(* CODESYS project SingleElevator.project

Project tree, tasks and I/O mapping:
  Device : CODESYS Control Win V3, 3S - Smart Software Solutions GmbH, version 3.5.12.20
    application Application
      libraries: Standard, * (System)
      task MainTask (cyclic, interval 30 ms, priority 1) calls Simulation, POU, GA_Collector
      task VISU_TASK (cyclic, interval 200 ms, priority 31) calls VisuElems.Visu_Prg
      program GA_Collector [FBD]
      global variables GVL
      program POU [SFC]: Doors_Closing_Homing_exit, Doors_Opening_Homing_exit, Homing_Motor_exit, Motor_Usage_active, Doors_Closing_active, Motor_Usage_exit, Doors_Opening_exit, Internal_Panel_exit, Internal_Panel_active, Doors_Closing_exit, Doors_Opening_active, Homing_Motor_active, Doors_Opening_Homing_active, Doors_Closing_Homing_active
      GAs/
        function block Doors_GA [SFC]: Ready_active, Busy_active
        function block Call_Management_GA [SFC]: Turn_Off_5_active, Refresh_dim_log_exit, P5_exit, Turn_Off_1_active, P2_active, P7_exit, Destination_Update_exit, Turn_Off_6_active, P3_exit, Destination_OUT_active, Wait_TIME_active, Ready_active, Ready_exit, P7_active, Turn_Off_G_active, WAIT_active, PG_active, Can_Go_active, P5_active, Sorting_Int_entry, Turn_Off_7_active, P6_exit, P6_active, Turn_Off_2_active, P2_exit, Turn_Off_4_active, Wait_Start_active, Waiting_Int_active, P1_exit, Wait_TIME_entry, P3_active, Destination_Update_active, P1_active, P4_active, Turn_Off_3_active, P4_exit, Refresh_dim_log_active, Turn_Off_Leds_active, Turn_Off_Leds_exit, Sorting_Int_active, Sorting_Int_exit, Waiting_Ext_active, Waiting_Int_entry, WAIT_entry, Turn_Off_3_exit, Sorting_Ext_entry, Sorting_Ext_active, Can_Go_exit, Turn_Off_Leds_entry, Control_Int_active, Wait_Passengers_exit
        function block Motor_GA [SFC]: Motor_Activation_DOWN_active, Ready_active, Wait_Arrive_Up_entry, Go_G_Deck_active, Deck_Passed_entry, Step1_active, Busy_active, Motor_Activation_Homing_active, Go_G_Deck_exit, Arrived_UP_exit, Arrived_Down_exit, Wait_Arrive_Up_exit, Motor_Activation_UP_active, Motor_Activation_Homing_exit, Wait_Arrive_Down_exit, Motor_Activation_Homing_entry, Wait_Arrive_Down_entry
      visualisation Visualization
      program Simulation [ST]
  text list GlobalTextList
*)

// Device/Application/GVL
VAR_GLOBAL
(* Elevator managing variables*)
	Open: BOOL;				(* Sensor: the door is fully open*)
	Closed: BOOL;			(* Sensor: the door is fully closed*)
	LimitDown: BOOL;		(* Sensor: lower limit sensor, if TRUE the lift has reached the lower limit*)
	LimitUp: BOOL;			(* Sensor: upper limit sensor, if TRUE the lift has reached the upper limit*)
	DeckSensor: BOOL;		(* Sensor: if TRUE the cab is in proximity of a deck*)
	RampSensor: BOOL;		(* Sensor: if TRUE the cab is in proximity of a ramp*)
	Presence :BOOL; 		(* Sensor: if TRUE something blocks the door photocell*)
	Emergency: BOOL;		(* Input: if TRUE the emergency button has been pressed*)

	Closing: BOOL;			(* Actuator: if TRUE the door starts closing*)
	Opening: BOOL;			(* Actuator: the door starts opening*)
	Motor_on: BOOL;			(* Actuator: if TRUE the lift pulley motor start moving*)
	Up: BOOL;				(* Actuator parameter: if TRUE the lift moves upward, downward otherwise*)
	Vel: BOOL;				(* Actuator parameter: motor speed, if TRUE high speed, low speed otherwise*)


	Current: INT;  			(* Visualization: variable used to storage the current deck*)
    Destination: INT;		(* Visualization: variable used to storage the the destination deck*)
	EmergencyVis: BOOL; 	(* Visualization: if TRUE the emergency light is turned on*)

	InitialDeck: INT := 1;	(* Only for simulation: variable used to define the initial deck*)
	InitCycle: BOOL := FALSE;(* Only for simulation: used to execute the instruction at the first cycle*)
	Height: INT;			(* Only for simulation: elevator height*)
	DeckRest: INT;        	(* Only for simulation: division rest for generating deck sensor*)
	Memory: INT;
	RampRest: INT;			(* Only for simulation: division rest for generating the ramp position*)
	MemoryR: INT;
	Door: INT;				(* Only for simulation: to visualize the closing of the door*)
	Displacement: INT;		(* Only for simulation: lift displacement, dependent on the motor speed*)

 (*Inputs: internal panel variables*)
	PG: BOOL;
	P1: BOOL;
	P2: BOOL;
	P3: BOOL;
	P4: BOOL;
	P5: BOOL;
	P6: BOOL;
	P7: BOOL;

(*Visualization: internal panel variables used to turn on the LED*)
	PGVis: BOOL;
	P1Vis: BOOL;
	P2Vis: BOOL;
	P3Vis: BOOL;
	P4Vis: BOOL;
	P5Vis: BOOL;
	P6Vis: BOOL;
	P7Vis: BOOL;

(*Inputs: external panel variables*)
	UpDeckG: BOOL;
	UpDeck1: BOOL;
	UpDeck2: BOOL;
	UpDeck3: BOOL;
	UpDeck4: BOOL;
	UpDeck5: BOOL;
	UpDeck6: BOOL;
	DownDeck7: BOOL;
	DownDeck6: BOOL;
	DownDeck5: BOOL;
	DownDeck4: BOOL;
	DownDeck3: BOOL;
	DownDeck2: BOOL;
	DownDeck1: BOOL;

(*Visualization: external panel variables used to turn on the LED*)
	UpDeckGVis: BOOL;
	UpDeck1Vis: BOOL;
	UpDeck2Vis: BOOL;
	UpDeck3Vis: BOOL;
	UpDeck4Vis: BOOL;
	UpDeck5Vis: BOOL;
	UpDeck6Vis: BOOL;
	DownDeck7Vis: BOOL;
	DownDeck6Vis: BOOL;
	DownDeck5Vis: BOOL;
	DownDeck4Vis: BOOL;
	DownDeck3Vis: BOOL;
	DownDeck2Vis: BOOL;
	DownDeck1Vis: BOOL;

(*Only for simulation: variables used to simulate the fault on deck sensor*)
	SensorG: BOOL;				(* if TRUE the magnetic information for deck G is lost and the deck sensor cannot become TRUE*)
	Sensor1: BOOL;				(* if TRUE the magnetic information for deck 1 is lost and the deck sensor cannot become TRUE*)
	Sensor2: BOOL;
	Sensor3: BOOL;
	Sensor4: BOOL;
	Sensor5: BOOL;
	Sensor6: BOOL;
	Sensor7: BOOL;
	FaultSensorAlarm: BOOL; 	(* Visulaization: if TRUE alerts the user of a deck sensor fault*)

(*Only for simulation: variables used to simulate the fault on ramp sensor*)
	RampGUp: BOOL;
	Ramp1Down: BOOL;
	Ramp1Up:BOOL;
	Ramp2Down: BOOL;
	Ramp2Up:BOOL;
	Ramp3Down: BOOL;
	Ramp3Up:BOOL;
	Ramp4Down: BOOL;
	Ramp4Up:BOOL;
	Ramp5Down: BOOL;
	Ramp5Up:BOOL;
	Ramp6Down: BOOL;
	Ramp6Up:BOOL;
	Ramp7Down: BOOL;
	FaultRampAlarm: BOOL; 		(* Visulaization: if TRUE alerts the user of a ramp sensor fault*)
	SensorGOK: BOOL;
	Sensor1OK: BOOL;
	Sensor2OK: BOOL;
	Sensor6OK: BOOL;
	Sensor3OK: BOOL;
	Sensor4OK: BOOL;
	Sensor5OK: BOOL;
	Sensor7OK: BOOL;
	RampGUpOK: BOOL;
	Ramp1DownOK: BOOL;
	Ramp1UpOK: BOOL;
	Ramp2DownOK: BOOL;
	Ramp2UpOK: BOOL;
	Ramp3DownOK: BOOL;
	Ramp3UpOK: BOOL;
	Ramp4DownOK: BOOL;
	Ramp4UpOK: BOOL;
	Ramp5DownOK: BOOL;
	Ramp5UpOK: BOOL;
	Ramp6DownOK: BOOL;
	Ramp6UpOK: BOOL;
	Ramp7DownOK: BOOL;
	Ramp7UpOK: BOOL;
	Doors: Doors_GA;
	Motor: Motor_GA;
	Call_Management: Call_Management_GA;
END_VAR

// Device/Application/Simulation
PROGRAM Simulation
VAR
END_VAR

(* Initial position of the cab inside the hoistway. It is executed only at the first cycle.  *)
IF NOT GVL.InitCycle THEN
			GVL.InitCycle := TRUE ;
			GVL.Height := 20 * GVL.InitialDeck;
		    GVL.Door := 0;
			GVL.Current := GVL.Height / 20;
END_IF;

(* Elevator management, these instructions are executed each cycle time*)

(* Elevator door control. *)
IF GVL.Closing THEN
	GVL.Door := GVL.Door + 1;		(*Closing door management*)
	GVL.Open := FALSE;
END_IF

IF GVL.Door >= 60 THEN						(* Closed door limit*)
	GVL.Closed := TRUE;
END_IF

IF GVL.Opening THEN
	GVL.Door := GVL.Door - 1; 	(* Opening door management*)
	GVL.Closed := FALSE;
END_IF

IF GVL.Door <= 0 THEN							(* Open door limit*)
	GVL.Open := TRUE;
END_IF


(* Maximum and minimum management in the door simulation*)
IF GVL.Door < 0 THEN
	 GVL.Door := 0;
END_IF

IF GVL.Door > 60 THEN
	GVL.Door := 60;
END_IF


(* Control of the cab position inside the hostway. *)
(* Displacement definition for graphic visualization*)
IF GVL.Vel THEN 
	GVL.Displacement := 2;
ELSE 
	GVL.Displacement := 1;
END_IF


(* Height modification relying on direction and speed*)
IF GVL.Motor_on AND GVL.Up THEN
	GVL.Height := GVL.Height + GVL.Displacement;
	GVL.LimitDown := FALSE;
END_IF

IF GVL.Motor_on AND NOT GVL.Up THEN
	GVL.Height := GVL.Height - GVL.Displacement;
	GVL.LimitUp := FALSE;
END_IF


(* Limits for visualization*)
IF GVL.Height < -20 THEN
	GVL.Height := -20;
END_IF

IF GVL.Height > 160 THEN
	GVL.Height := 160;
END_IF

(* Limit sensors management*)
IF GVL.Height <= -10 THEN
	GVL.LimitDown := TRUE;
END_IF

IF GVL.Height >= 150 THEN
	 GVL.LimitUp := TRUE;
END_IF


(*-------------------------------------------------------------------*)
(*  Fault Management (Deck and Ramp Sensors)   *)
(*-------------------------------------------------------------------*)
(* Deck Sensor*)
(* Range of value where the deck sensor is active*)
IF ((GVL.Height >= -1) AND (GVL.Height <= 1)) THEN
	GVL.SensorGOK := TRUE;
ELSE  
	GVL.SensorGOK := FALSE;
END_IF

IF ((GVL.Height >= 20-1) AND (GVL.Height <= 20+1)) THEN
	GVL.Sensor1OK := TRUE;
ELSE  
	GVL.Sensor1OK := FALSE;
END_IF

IF ((GVL.Height >= 40-1) AND (GVL.Height <= 40+1)) THEN
	GVL.Sensor2OK := TRUE;
ELSE  
	GVL.Sensor2OK := FALSE;
END_IF

IF ((GVL.Height >= 60-1) AND (GVL.Height <= 60+1)) THEN
	GVL.Sensor3OK := TRUE;
ELSE  
	GVL.Sensor3OK := FALSE;
END_IF

IF ((GVL.Height >= 80-1) AND (GVL.Height <= 80+1)) THEN
	GVL.Sensor4OK := TRUE;
ELSE  
	GVL.Sensor4OK := FALSE;
END_IF

IF ((GVL.Height >= 100-1) AND (GVL.Height <= 100+1)) THEN
	GVL.Sensor5OK := TRUE;
ELSE   
	GVL.Sensor5OK := FALSE;
END_IF

IF ((GVL.Height >= 120-1) AND (GVL.Height <= 120+1)) THEN
	GVL.Sensor6OK := TRUE;
ELSE  
	GVL.Sensor6OK := FALSE;
END_IF

IF ((GVL.Height >= 140-1) AND (GVL.Height <= 140+1)) THEN
	GVL.Sensor7OK := TRUE;
ELSE  
	GVL.Sensor7OK := FALSE;
END_IF

GVL.DeckSensor := (GVL.SensorGOK AND NOT GVL.SensorG) OR
				    (GVL.Sensor1OK AND NOT GVL.Sensor1) OR
				    (GVL.Sensor2OK AND NOT GVL.Sensor2) OR
				    (GVL.Sensor3OK AND NOT GVL.Sensor3) OR
				    (GVL.Sensor4OK AND NOT GVL.Sensor4) OR
				    (GVL.Sensor5OK AND NOT GVL.Sensor5) OR
				    (GVL.Sensor6OK AND NOT GVL.Sensor6) OR
				    (GVL.Sensor7OK AND NOT GVL.Sensor7);

(* Ramp Sensor*)
(* Range of value where the ramp sensor is active*)
IF ((GVL.Height >= 5-1) AND (GVL.Height <= 5+1)) THEN
	GVL.RampGUpOK := TRUE;
ELSE 
	GVL.RampGUpOK := FALSE;
END_IF

(* Ramp close to deck 1*)
IF ((GVL.Height >= 15-1) AND (GVL.Height <= 15+1)) THEN
	GVL.Ramp1DownOK := TRUE;
ELSE 
	GVL.Ramp1DownOK := FALSE;
END_IF

IF ((GVL.Height >= 25-1) AND (GVL.Height <= 25+1)) THEN
	GVL.Ramp1UpOK := TRUE;
ELSE 
	GVL.Ramp1UpOK := FALSE;
END_IF

(* Ramp close to deck 2*)
IF ((GVL.Height >= 35-1) AND (GVL.Height <= 35+1)) THEN
	GVL.Ramp2DownOK := TRUE;
ELSE 
	GVL.Ramp2DownOK := FALSE;
END_IF

IF ((GVL.Height >= 45-1) AND (GVL.Height <= 45+1)) THEN
	GVL.Ramp2UpOK := TRUE;
ELSE 
	GVL.Ramp2UpOK := FALSE;
END_IF

(*Ramp close to deck  3*)
IF ((GVL.Height >= 55-1) AND (GVL.Height <= 55+1)) THEN
	GVL.Ramp3DownOK := TRUE;
ELSE 
	GVL.Ramp3DownOK := FALSE;
END_IF

IF ((GVL.Height >= 65-1) AND (GVL.Height <= 65+1)) THEN
	GVL.Ramp3UpOK := TRUE;
ELSE 
	GVL.Ramp3UpOK := FALSE;
END_IF

(* Ramp close to deck  4*)
IF ((GVL.Height >= 75-1) AND (GVL.Height <= 75+1)) THEN
	GVL.Ramp4DownOK := TRUE;
ELSE 
	GVL.Ramp4DownOK := FALSE;
END_IF

IF ((GVL.Height >= 85-1) AND (GVL.Height <= 85+1)) THEN
	GVL.Ramp4UpOK := TRUE;
ELSE 
	GVL.Ramp4UpOK:=FALSE;
END_IF

(* Ramp close to deck  5*)
IF ((GVL.Height >= 95-1) AND (GVL.Height <= 95+1)) THEN
	GVL.Ramp5DownOK := TRUE;
ELSE 
	GVL.Ramp5DownOK := FALSE;
END_IF

IF ((GVL.Height >= 105-1) AND (GVL.Height <= 105+1)) THEN
	GVL.Ramp5UpOK := TRUE;
ELSE
	GVL.Ramp5UpOK := FALSE;
END_IF

(* Ramp close to deck  6*)
IF ((GVL.Height >= 115-1) AND (GVL.Height <= 115+1)) THEN
	GVL.Ramp6DownOK := TRUE;
ELSE 
	GVL.Ramp6DownOK := FALSE;
END_IF

IF ((GVL.Height >= 125-1) AND (GVL.Height <= 125+1)) THEN
	GVL.Ramp6UpOK := TRUE;
ELSE 
	GVL.Ramp6UpOK := FALSE;
END_IF

(* Ramp close to deck  7*)
IF ((GVL.Height >= 135-1) AND (GVL.Height <= 135+1)) THEN
	GVL.Ramp7DownOK := TRUE;
ELSE 
	GVL.Ramp7DownOK := FALSE;
END_IF

GVL.RampSensor:=(GVL.RampGUpOK AND NOT GVL.RampGUp) OR 
								(GVL.Ramp1DownOK AND NOT GVL.Ramp1Down ) OR 
								(GVL.Ramp1UpOK AND NOT GVL.Ramp1Up ) OR
								(GVL.Ramp2DownOK AND NOT GVL.Ramp2Down ) OR 
								(GVL.Ramp2UpOK AND NOT GVL.Ramp2Up ) OR
								(GVL.Ramp3DownOK AND NOT GVL.Ramp3Down ) OR
 								(GVL.Ramp3UpOK AND NOT GVL.Ramp3Up ) OR
								(GVL.Ramp4DownOK AND NOT GVL.Ramp4Down ) OR
 								(GVL.Ramp4UpOK AND NOT GVL.Ramp4Up ) OR
								(GVL.Ramp5DownOK AND NOT GVL.Ramp5Down ) OR
 								(GVL.Ramp5UpOK AND NOT GVL.Ramp5Up ) OR
								(GVL.Ramp6DownOK AND NOT GVL.Ramp6Down ) OR
								(GVL.Ramp6UpOK AND NOT GVL.Ramp6Up ) OR
								(GVL.Ramp7DownOK AND NOT GVL.Ramp7Down );

END_PROGRAM

// Device/Application/POU
PROGRAM POU
VAR
	Operation_OK: BOOL;
	Synchronization : BOOL;
END_VAR

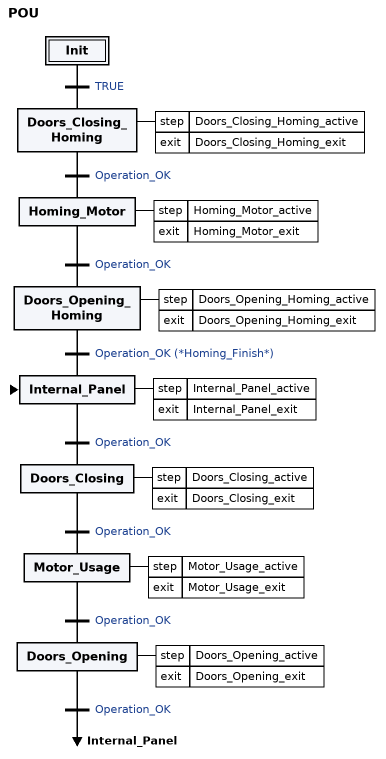
INITIAL_STEP Init:
END_STEP
TRANSITION FROM Init TO Doors_Closing_Homing
    := TRUE;
END_TRANSITION
STEP Doors_Closing_Homing:
    Doors_Closing_Homing_active(N);  // step action
    Doors_Closing_Homing_exit(P0);  // exit action
END_STEP
TRANSITION FROM Doors_Closing_Homing TO Homing_Motor
    := Operation_OK;
END_TRANSITION
STEP Homing_Motor:
    Homing_Motor_active(N);  // step action
    Homing_Motor_exit(P0);  // exit action
END_STEP
TRANSITION FROM Homing_Motor TO Doors_Opening_Homing
    := Operation_OK;
END_TRANSITION
STEP Doors_Opening_Homing:
    Doors_Opening_Homing_active(N);  // step action
    Doors_Opening_Homing_exit(P0);  // exit action
END_STEP
TRANSITION FROM Doors_Opening_Homing TO Internal_Panel
    := Operation_OK (*Homing_Finish*);
END_TRANSITION
STEP Internal_Panel:
    Internal_Panel_active(N);  // step action
    Internal_Panel_exit(P0);  // exit action
END_STEP
TRANSITION FROM Internal_Panel TO Doors_Closing
    := Operation_OK;
END_TRANSITION
STEP Doors_Closing:
    Doors_Closing_active(N);  // step action
    Doors_Closing_exit(P0);  // exit action
END_STEP
TRANSITION FROM Doors_Closing TO Motor_Usage
    := Operation_OK;
END_TRANSITION
STEP Motor_Usage:
    Motor_Usage_active(N);  // step action
    Motor_Usage_exit(P0);  // exit action
END_STEP
TRANSITION FROM Motor_Usage TO Doors_Opening
    := Operation_OK;
END_TRANSITION
STEP Doors_Opening:
    Doors_Opening_active(N);  // step action
    Doors_Opening_exit(P0);  // exit action
END_STEP
TRANSITION FROM Doors_Opening TO Internal_Panel
    := Operation_OK;
END_TRANSITION

ACTION Doors_Closing_Homing_exit:
Operation_OK:=FALSE;
Synchronization:=FALSE;
END_ACTION

ACTION Doors_Opening_Homing_exit:
Operation_OK:=FALSE;
Synchronization:=FALSE;
END_ACTION

ACTION Homing_Motor_exit:
Operation_OK:=FALSE;
Synchronization:=FALSE;
END_ACTION

ACTION Motor_Usage_active:
IF Motor.State = 'Ready' THEN
	Motor.Do_:= TRUE;
	Motor.STOP := FALSE;
	IF ( Call_Management.Destination_Deck[0] > Current AND Call_Management.Destination_Deck[0] <> 8 ) THEN
		Motor.Do_What := 'Go_Up';
	END_IF
	IF ( Call_Management.Destination_Deck[0] < Current AND Call_Management.Destination_Deck[0] <> 8 ) THEN
		Motor.Do_What := 'Go_Down';
	END_IF
END_IF

IF (Motor.State = 'Busy' AND Current = Call_Management.Destination_Deck [0] - 1 AND Motor.Do_What = 'Go_Up' OR Call_Management.Destination_Deck [0] = 8 ) THEN;
	Motor.STOP := TRUE;	
END_IF

IF (Motor.State = 'Busy' AND Current = Call_Management.Destination_Deck [0] + 1 AND Motor.Do_What = 'Go_Down' OR Call_Management.Destination_Deck [0] = 8 ) THEN;
	Motor.STOP := TRUE;	
END_IF

IF Motor.State = 'Busy' AND Motor.Done = TRUE THEN
	Motor.Do_ := FALSE;
	Motor.STOP := FALSE;
	Synchronization := TRUE;
END_IF

Operation_OK := Synchronization AND NOT Motor.Done;
END_ACTION

ACTION Doors_Closing_active:
IF Doors.State = 'Ready' THEN
	Doors.Do_:= TRUE;
	Doors.Do_what := 'Close';
END_IF

IF Doors.State = 'Busy' AND Doors.Done = TRUE THEN
	Doors.Do_ := FALSE;
	Synchronization := TRUE;
END_IF

Operation_OK := Synchronization AND NOT Doors.Done;
END_ACTION

ACTION Motor_Usage_exit:
Operation_OK:=FALSE;
Synchronization:=FALSE;
END_ACTION

ACTION Doors_Opening_exit:
Operation_OK:=FALSE;
Synchronization:=FALSE;
END_ACTION

ACTION Internal_Panel_exit:
Operation_OK:=FALSE;
Synchronization:=FALSE;
END_ACTION

ACTION Internal_Panel_active:
IF Call_Management.State = 'Ready' THEN
	Call_Management.Start:= TRUE;
	Call_Management.Stop:= FALSE;
END_IF

IF Call_Management.State = 'Can_Go' THEN
	Synchronization := TRUE;
END_IF

Operation_OK := Synchronization;
END_ACTION

ACTION Doors_Closing_exit:
Operation_OK:=FALSE;
Synchronization:=FALSE;
END_ACTION

ACTION Doors_Opening_active:
IF Doors.State = 'Ready' THEN
	Doors.Do_:= TRUE;
	Doors.Do_what := 'Open';
END_IF

IF Doors.State = 'Busy' AND Doors.Done = TRUE AND Call_Management.Destination_Deck[0] <> 8 THEN
	Doors.Do_ := FALSE;
	Synchronization := TRUE;
END_IF

Operation_OK := Synchronization AND NOT Doors.Done;
END_ACTION

ACTION Homing_Motor_active:
IF Motor.State = 'Ready' THEN
	Motor.Do_:= TRUE;
	Motor.Do_What := 'Homing';
END_IF

IF Motor.State = 'Busy' AND Motor.Done = TRUE THEN
	Motor.Do_ := FALSE;
	Synchronization := TRUE;
END_IF

Operation_OK := Synchronization AND NOT Motor.Done;
END_ACTION

ACTION Doors_Opening_Homing_active:
IF Doors.State = 'Ready' THEN
	Doors.Do_:= TRUE;
	Doors.Do_what := 'Open';
END_IF

IF Doors.State = 'Busy' AND Doors.Done = TRUE THEN
	Doors.Do_ := FALSE;
	Synchronization := TRUE;
END_IF

Operation_OK := Synchronization AND NOT Doors.Done;
END_ACTION

ACTION Doors_Closing_Homing_active:
IF Doors.State = 'Ready' THEN
	Doors.Do_:= TRUE;
	Doors.Do_what := 'Close';
END_IF

IF Doors.State = 'Busy' AND Doors.Done = TRUE THEN
	Doors.Do_ := FALSE;
	Synchronization := TRUE;
END_IF

Operation_OK := Synchronization AND NOT Doors.Done;
END_ACTION

END_PROGRAM

// Device/Application/GA_Collector
PROGRAM GA_Collector
VAR
END_VAR

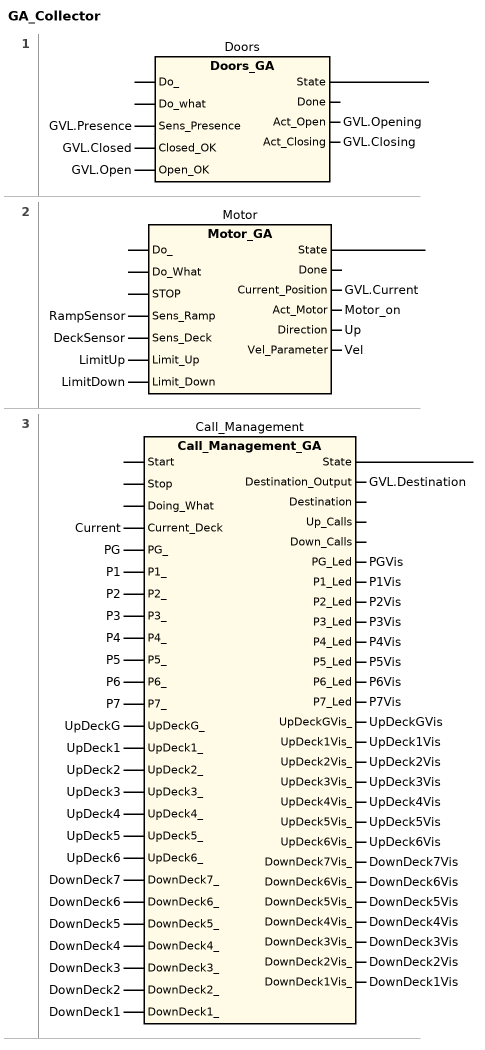
// NETWORK 1
Doors(
    Sens_Presence := GVL.Presence,
    Closed_OK := GVL.Closed,
    Open_OK := GVL.Open,
    Act_Open => GVL.Opening,
    Act_Closing => GVL.Closing); // Doors_GA

// NETWORK 2
Motor(
    Sens_Ramp := RampSensor,
    Sens_Deck := DeckSensor,
    Limit_Up := LimitUp,
    Limit_Down := LimitDown,
    Current_Position => GVL.Current,
    Act_Motor => Motor_on,
    Direction => Up,
    Vel_Parameter => Vel); // Motor_GA

// NETWORK 3
Call_Management(
    Current_Deck := Current,
    PG_ := PG,
    P1_ := P1,
    P2_ := P2,
    P3_ := P3,
    P4_ := P4,
    P5_ := P5,
    P6_ := P6,
    P7_ := P7,
    UpDeckG_ := UpDeckG,
    UpDeck1_ := UpDeck1,
    UpDeck2_ := UpDeck2,
    UpDeck3_ := UpDeck3,
    UpDeck4_ := UpDeck4,
    UpDeck5_ := UpDeck5,
    UpDeck6_ := UpDeck6,
    DownDeck7_ := DownDeck7,
    DownDeck6_ := DownDeck6,
    DownDeck5_ := DownDeck5,
    DownDeck4_ := DownDeck4,
    DownDeck3_ := DownDeck3,
    DownDeck2_ := DownDeck2,
    DownDeck1_ := DownDeck1,
    Destination_Output => GVL.Destination,
    PG_Led => PGVis,
    P1_Led => P1Vis,
    P2_Led => P2Vis,
    P3_Led => P3Vis,
    P4_Led => P4Vis,
    P5_Led => P5Vis,
    P6_Led => P6Vis,
    P7_Led => P7Vis,
    UpDeckGVis_ => UpDeckGVis,
    UpDeck1Vis_ => UpDeck1Vis,
    UpDeck2Vis_ => UpDeck2Vis,
    UpDeck3Vis_ => UpDeck3Vis,
    UpDeck4Vis_ => UpDeck4Vis,
    UpDeck5Vis_ => UpDeck5Vis,
    UpDeck6Vis_ => UpDeck6Vis,
    DownDeck7Vis_ => DownDeck7Vis,
    DownDeck6Vis_ => DownDeck6Vis,
    DownDeck5Vis_ => DownDeck5Vis,
    DownDeck4Vis_ => DownDeck4Vis,
    DownDeck3Vis_ => DownDeck3Vis,
    DownDeck2Vis_ => DownDeck2Vis,
    DownDeck1Vis_ => DownDeck1Vis); // Call_Management_GA

END_PROGRAM

// Device/Application/GAs/Doors_GA
FUNCTION_BLOCK Doors_GA
VAR_INPUT
	Do_: BOOL;
	Do_what: STRING;
	Sens_Presence: BOOL;
	Closed_OK: BOOL;
	Open_OK: BOOL;
END_VAR
VAR_OUTPUT
	State: STRING;
	Done: BOOL;
	Act_Open: BOOL;
	Act_Closing: BOOL;
END_VAR
VAR	
END_VAR

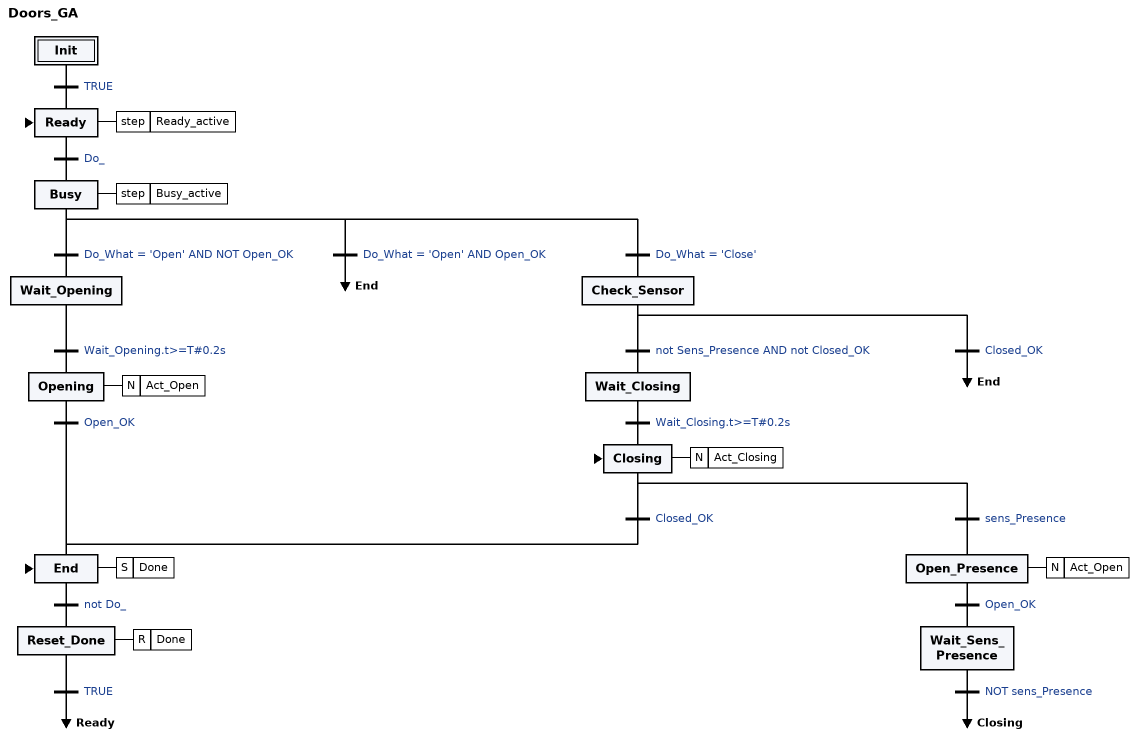
INITIAL_STEP Init:
END_STEP
TRANSITION FROM Init TO Ready
    := TRUE;
END_TRANSITION
STEP Ready:
    Ready_active(N);  // step action
END_STEP
TRANSITION FROM Ready TO Busy
    := Do_;
END_TRANSITION
STEP Busy:
    Busy_active(N);  // step action
END_STEP
TRANSITION FROM Busy TO Wait_Opening
    := Do_What = 'Open' AND NOT Open_OK;
END_TRANSITION
STEP Wait_Opening:
END_STEP
TRANSITION FROM Wait_Opening TO Opening
    := Wait_Opening.t>=T#0.2s;
END_TRANSITION
STEP Opening:
    Act_Open(N);
END_STEP
TRANSITION FROM Opening TO End
    := Open_OK;
END_TRANSITION
TRANSITION FROM Busy TO End
    := Do_What = 'Open' AND Open_OK;
END_TRANSITION
TRANSITION FROM Busy TO Check_Sensor
    := Do_What = 'Close';
END_TRANSITION
STEP Check_Sensor:
END_STEP
TRANSITION FROM Check_Sensor TO Wait_Closing
    := not Sens_Presence AND not Closed_OK;
END_TRANSITION
STEP Wait_Closing:
END_STEP
TRANSITION FROM Wait_Closing TO Closing
    := Wait_Closing.t>=T#0.2s;
END_TRANSITION
STEP Closing:
    Act_Closing(N);
END_STEP
TRANSITION FROM Closing TO End
    := Closed_OK;
END_TRANSITION
TRANSITION FROM Closing TO Open_Presence
    := sens_Presence;
END_TRANSITION
STEP Open_Presence:
    Act_Open(N);
END_STEP
TRANSITION FROM Open_Presence TO Wait_Sens_Presence
    := Open_OK;
END_TRANSITION
STEP Wait_Sens_Presence:
END_STEP
TRANSITION FROM Wait_Sens_Presence TO Closing
    := NOT sens_Presence;
END_TRANSITION
TRANSITION FROM Check_Sensor TO End
    := Closed_OK;
END_TRANSITION
STEP End:
    Done(S);
END_STEP
TRANSITION FROM End TO Reset_Done
    := not Do_;
END_TRANSITION
STEP Reset_Done:
    Done(R);
END_STEP
TRANSITION FROM Reset_Done TO Ready
    := TRUE;
END_TRANSITION

ACTION Ready_active:
State := 'Ready';
END_ACTION

ACTION Busy_active:
State := 'Busy';
END_ACTION

END_FUNCTION_BLOCK

// Device/Application/GAs/Motor_GA
FUNCTION_BLOCK Motor_GA
VAR_INPUT
	Do_ : BOOL;
	Do_What: STRING;
	STOP: BOOL;
	Sens_Ramp: BOOL;
	Sens_Deck: BOOL;
	Limit_Up: BOOL;
	Limit_Down: BOOL;
END_VAR
VAR_OUTPUT
	State : STRING;
	Done : BOOL;
	Current_Position : INT;
	Act_Motor: BOOL;
	Direction: BOOL;
	Vel_Parameter: BOOL;
END_VAR
VAR
END_VAR

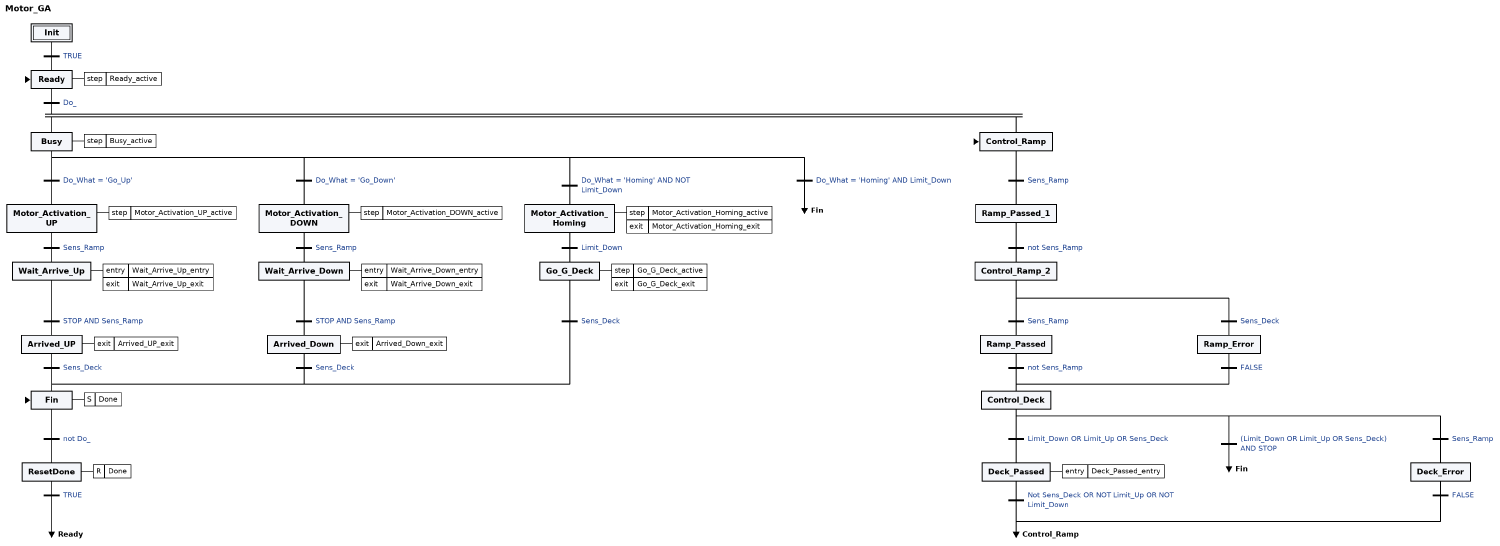
INITIAL_STEP Init:
END_STEP
TRANSITION FROM Init TO Ready
    := TRUE;
END_TRANSITION
STEP Ready:
    Ready_active(N);  // step action
END_STEP
TRANSITION FROM Ready TO (Busy, Control_Ramp)
    := Do_;
END_TRANSITION
STEP Busy:
    Busy_active(N);  // step action
END_STEP
TRANSITION FROM Busy TO Motor_Activation_UP
    := Do_What = 'Go_Up';
END_TRANSITION
STEP Motor_Activation_UP:
    Motor_Activation_UP_active(N);  // step action
END_STEP
TRANSITION FROM Motor_Activation_UP TO Wait_Arrive_Up
    := Sens_Ramp;
END_TRANSITION
STEP Wait_Arrive_Up:
    Wait_Arrive_Up_entry(P1);  // entry action
    Wait_Arrive_Up_exit(P0);  // exit action
END_STEP
TRANSITION FROM Wait_Arrive_Up TO Arrived_UP
    := STOP AND Sens_Ramp;
END_TRANSITION
STEP Arrived_UP:
    Arrived_UP_exit(P0);  // exit action
END_STEP
TRANSITION FROM Arrived_UP TO Fin
    := Sens_Deck;
END_TRANSITION
TRANSITION FROM Busy TO Motor_Activation_DOWN
    := Do_What = 'Go_Down';
END_TRANSITION
STEP Motor_Activation_DOWN:
    Motor_Activation_DOWN_active(N);  // step action
END_STEP
TRANSITION FROM Motor_Activation_DOWN TO Wait_Arrive_Down
    := Sens_Ramp;
END_TRANSITION
STEP Wait_Arrive_Down:
    Wait_Arrive_Down_entry(P1);  // entry action
    Wait_Arrive_Down_exit(P0);  // exit action
END_STEP
TRANSITION FROM Wait_Arrive_Down TO Arrived_Down
    := STOP AND Sens_Ramp;
END_TRANSITION
STEP Arrived_Down:
    Arrived_Down_exit(P0);  // exit action
END_STEP
TRANSITION FROM Arrived_Down TO Fin
    := Sens_Deck;
END_TRANSITION
TRANSITION FROM Busy TO Motor_Activation_Homing
    := Do_What = 'Homing' AND NOT Limit_Down;
END_TRANSITION
STEP Motor_Activation_Homing:
    Motor_Activation_Homing_active(N);  // step action
    Motor_Activation_Homing_exit(P0);  // exit action
END_STEP
TRANSITION FROM Busy TO Fin
    := Do_What = 'Homing' AND Limit_Down;
END_TRANSITION
TRANSITION FROM Motor_Activation_Homing TO Go_G_Deck
    := Limit_Down;
END_TRANSITION
STEP Go_G_Deck:
    Go_G_Deck_active(N);  // step action
    Go_G_Deck_exit(P0);  // exit action
END_STEP
TRANSITION FROM Go_G_Deck TO Fin
    := Sens_Deck;
END_TRANSITION
STEP Fin:
    Done(S);
END_STEP
STEP Control_Ramp:
END_STEP
TRANSITION FROM Control_Ramp TO Ramp_Passed_1
    := Sens_Ramp;
END_TRANSITION
STEP Ramp_Passed_1:
END_STEP
TRANSITION FROM Ramp_Passed_1 TO Control_Ramp_2
    := not Sens_Ramp;
END_TRANSITION
STEP Control_Ramp_2:
END_STEP
TRANSITION FROM Control_Ramp_2 TO Ramp_Passed
    := Sens_Ramp;
END_TRANSITION
STEP Ramp_Passed:
END_STEP
TRANSITION FROM Ramp_Passed TO Control_Deck
    := not Sens_Ramp;
END_TRANSITION
TRANSITION FROM Control_Ramp_2 TO Ramp_Error
    := Sens_Deck;
END_TRANSITION
STEP Ramp_Error:
END_STEP
TRANSITION FROM Ramp_Error TO Control_Deck
    := FALSE;
END_TRANSITION
STEP Control_Deck:
END_STEP
TRANSITION FROM Control_Deck TO Deck_Passed
    := Limit_Down OR Limit_Up OR Sens_Deck;
END_TRANSITION
STEP Deck_Passed:
    Deck_Passed_entry(P1);  // entry action
END_STEP
TRANSITION FROM Deck_Passed TO Control_Ramp
    := Not Sens_Deck OR NOT Limit_Up OR NOT Limit_Down;
END_TRANSITION
TRANSITION FROM Control_Deck TO Fin
    := (Limit_Down OR Limit_Up OR Sens_Deck) AND STOP;
END_TRANSITION
TRANSITION FROM Control_Deck TO Deck_Error
    := Sens_Ramp;
END_TRANSITION
STEP Deck_Error:
END_STEP
TRANSITION FROM Deck_Error TO Control_Ramp
    := FALSE;
END_TRANSITION
TRANSITION FROM Fin TO ResetDone
    := not Do_;
END_TRANSITION
STEP ResetDone:
    Done(R);
END_STEP
TRANSITION FROM ResetDone TO Ready
    := TRUE;
END_TRANSITION
// branch label Fault

ACTION Motor_Activation_DOWN_active:
Act_Motor := TRUE;
END_ACTION

ACTION Ready_active:
State := 'Ready';
END_ACTION

ACTION Wait_Arrive_Up_entry:
Vel_Parameter := TRUE;
END_ACTION

ACTION Go_G_Deck_active:
Current_Position := -1;
Direction:= TRUE;
END_ACTION

ACTION Deck_Passed_entry:
IF Do_What = 'Go_Up' AND Act_Motor THEN
	Current_Position := Current_Position +1;
END_IF

IF Do_What = 'Go_Down' AND Act_Motor THEN
	Current_Position := Current_Position -1;
END_IF
END_ACTION

ACTION Step1_active:
Current_Position := Current_Position +1;
END_ACTION

ACTION Busy_active:
State := 'Busy';
END_ACTION

ACTION Motor_Activation_Homing_active:
Act_Motor := TRUE;
(* La simulazione ha gia impostato all'interno di settare il current a -1 *)
END_ACTION

ACTION Go_G_Deck_exit:
Act_Motor := FALSE;
END_ACTION

ACTION Arrived_UP_exit:
Act_Motor := FALSE;
Direction := FALSE;
Current_Position := Current_Position +1;
END_ACTION

ACTION Arrived_Down_exit:
Act_Motor := FALSE;
Direction := FALSE;
Current_Position:= Current_Position -1;
END_ACTION

ACTION Wait_Arrive_Up_exit:
Vel_Parameter := FALSE;
END_ACTION

ACTION Motor_Activation_UP_active:
Act_Motor := TRUE;
Direction := TRUE;
END_ACTION

ACTION Motor_Activation_Homing_exit:
Current_Position := -1;
END_ACTION

ACTION Wait_Arrive_Down_exit:
Vel_Parameter := FALSE;
END_ACTION

ACTION Motor_Activation_Homing_entry:
Current_Position := 1;
END_ACTION

ACTION Wait_Arrive_Down_entry:
Vel_Parameter := TRUE;
END_ACTION

END_FUNCTION_BLOCK

// Device/Application/GAs/Call_Management_GA
FUNCTION_BLOCK Call_Management_GA
VAR_INPUT
	Start : BOOL;
	Stop: BOOL;
	Doing_What : STRING;
	Current_Deck : INT;
	PG_: BOOL; 
	P1_: BOOL;
	P2_: BOOL;
	P3_: BOOL;
	P4_: BOOL;
	P5_: BOOL;
	P6_: BOOL;
	P7_: BOOL;
	UpDeckG_: BOOL;
	UpDeck1_: BOOL;
	UpDeck2_: BOOL;
	UpDeck3_: BOOL;
	UpDeck4_: BOOL;
	UpDeck5_: BOOL;
	UpDeck6_: BOOL;
	DownDeck7_: BOOL;
	DownDeck6_: BOOL;
	DownDeck5_: BOOL;
	DownDeck4_: BOOL;
	DownDeck3_: BOOL;
	DownDeck2_: BOOL;
	DownDeck1_: BOOL;
END_VAR
VAR_OUTPUT
	State : STRING;
	Destination_Output : INT;
	Destination_Deck : ARRAY [0..7] OF INT := [8(8)];
	Up_Calls : ARRAY [0..13] OF INT := [14(8)];
	Down_Calls : ARRAY [0..13] OF INT := [14(8)];
	PG_Led: BOOL;
	P1_Led: BOOL;
	P2_Led: BOOL;
	P3_Led: BOOL;
	P4_Led: BOOL;
	P5_Led: BOOL;
	P6_Led: BOOL;
	P7_Led: BOOL;
	UpDeckGVis_: BOOL;
	UpDeck1Vis_: BOOL;
	UpDeck2Vis_: BOOL;
	UpDeck3Vis_: BOOL;
	UpDeck4Vis_: BOOL;
	UpDeck5Vis_: BOOL;
	UpDeck6Vis_: BOOL;
	DownDeck7Vis_: BOOL;
	DownDeck6Vis_: BOOL;
	DownDeck5Vis_: BOOL;
	DownDeck4Vis_: BOOL;
	DownDeck3Vis_: BOOL;
	DownDeck2Vis_: BOOL;
	DownDeck1Vis_: BOOL;
END_VAR
VAR
	{*INTERNAL PANEL SORT*}
	i : INT := 0;
	dim_cabin: INT :=0;
	j: INT;
	Sorted: BOOL;
	t: INT;
	
	{*EXTERNAL PANEL*}
	ext: INT :=0;
	z: INT;
	Position_Ext: INT :=8;
	
	k: INT :=0;
	Served: BOOL;
	
	Turned_Off: BOOL;
	Pressed_Int: BOOL;
	Pressed_Start: BOOL;
	
	g: INT;
	Finish: BOOL;
	Upgrading: BOOL;
	Upgraded: BOOL;
END_VAR

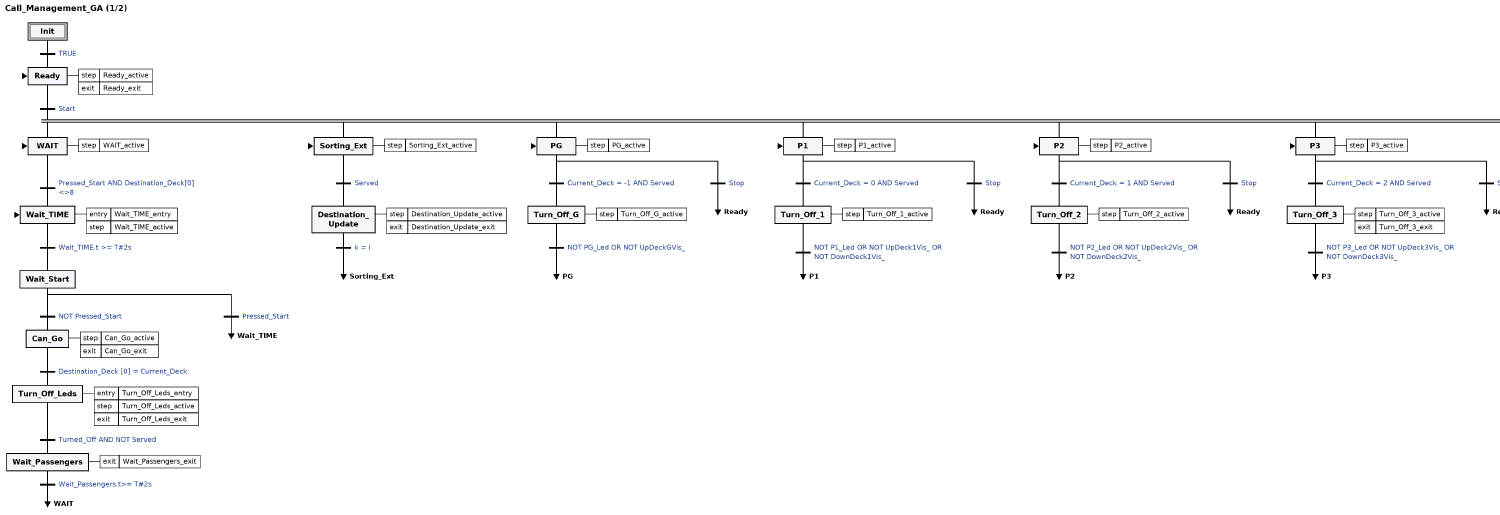
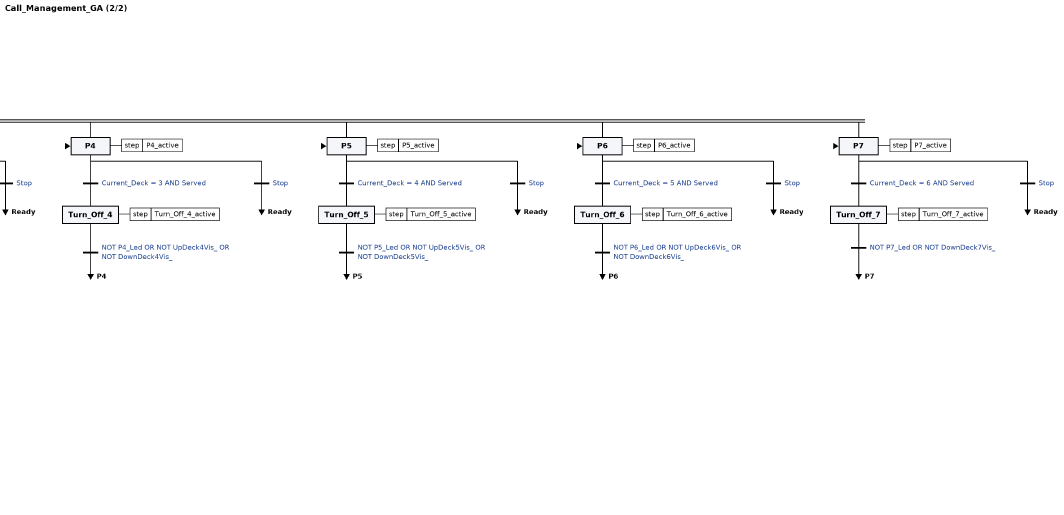
INITIAL_STEP Init:
END_STEP
TRANSITION FROM Init TO Ready
    := TRUE;
END_TRANSITION
STEP Ready:
    Ready_active(N);  // step action
    Ready_exit(P0);  // exit action
END_STEP
TRANSITION FROM Ready TO (WAIT, Sorting_Ext, PG, P1, P2, P3, P4, P5, P6, P7)
    := Start;
END_TRANSITION
STEP WAIT:
    WAIT_active(N);  // step action
END_STEP
TRANSITION FROM WAIT TO Wait_TIME
    := Pressed_Start AND Destination_Deck[0] <>8;
END_TRANSITION
STEP Wait_TIME:
    Wait_TIME_entry(P1);  // entry action
    Wait_TIME_active(N);  // step action
END_STEP
TRANSITION FROM Wait_TIME TO Wait_Start
    := Wait_TIME.t >= T#2s;
END_TRANSITION
STEP Wait_Start:
END_STEP
TRANSITION FROM Wait_Start TO Can_Go
    := NOT Pressed_Start;
END_TRANSITION
TRANSITION FROM Wait_Start TO Wait_TIME
    := Pressed_Start;
END_TRANSITION
STEP Can_Go:
    Can_Go_active(N);  // step action
    Can_Go_exit(P0);  // exit action
END_STEP
TRANSITION FROM Can_Go TO Turn_Off_Leds
    := Destination_Deck [0] = Current_Deck;
END_TRANSITION
STEP Turn_Off_Leds:
    Turn_Off_Leds_entry(P1);  // entry action
    Turn_Off_Leds_active(N);  // step action
    Turn_Off_Leds_exit(P0);  // exit action
END_STEP
TRANSITION FROM Turn_Off_Leds TO Wait_Passengers
    := Turned_Off AND NOT Served;
END_TRANSITION
STEP Wait_Passengers:
    Wait_Passengers_exit(P0);  // exit action
END_STEP
TRANSITION FROM Wait_Passengers TO WAIT
    := Wait_Passengers.t>= T#2s;
END_TRANSITION
STEP Sorting_Ext:
    Sorting_Ext_active(N);  // step action
END_STEP
TRANSITION FROM Sorting_Ext TO Destination_Update
    := Served;
END_TRANSITION
STEP Destination_Update:
    Destination_Update_active(N);  // step action
    Destination_Update_exit(P0);  // exit action
END_STEP
TRANSITION FROM Destination_Update TO Sorting_Ext
    := k = i;
END_TRANSITION
STEP PG:
    PG_active(N);  // step action
END_STEP
TRANSITION FROM PG TO Turn_Off_G
    := Current_Deck = -1 AND Served;
END_TRANSITION
STEP Turn_Off_G:
    Turn_Off_G_active(N);  // step action
END_STEP
TRANSITION FROM Turn_Off_G TO PG
    := NOT PG_Led OR NOT UpDeckGVis_;
END_TRANSITION
TRANSITION FROM PG TO Ready
    := Stop;
END_TRANSITION
STEP P1:
    P1_active(N);  // step action
END_STEP
TRANSITION FROM P1 TO Turn_Off_1
    := Current_Deck = 0 AND Served;
END_TRANSITION
STEP Turn_Off_1:
    Turn_Off_1_active(N);  // step action
END_STEP
TRANSITION FROM Turn_Off_1 TO P1
    := NOT P1_Led OR NOT UpDeck1Vis_ OR NOT DownDeck1Vis_;
END_TRANSITION
TRANSITION FROM P1 TO Ready
    := Stop;
END_TRANSITION
STEP P2:
    P2_active(N);  // step action
END_STEP
TRANSITION FROM P2 TO Turn_Off_2
    := Current_Deck = 1 AND Served;
END_TRANSITION
STEP Turn_Off_2:
    Turn_Off_2_active(N);  // step action
END_STEP
TRANSITION FROM Turn_Off_2 TO P2
    := NOT P2_Led OR NOT UpDeck2Vis_ OR NOT DownDeck2Vis_;
END_TRANSITION
TRANSITION FROM P2 TO Ready
    := Stop;
END_TRANSITION
STEP P3:
    P3_active(N);  // step action
END_STEP
TRANSITION FROM P3 TO Turn_Off_3
    := Current_Deck = 2 AND Served;
END_TRANSITION
STEP Turn_Off_3:
    Turn_Off_3_active(N);  // step action
    Turn_Off_3_exit(P0);  // exit action
END_STEP
TRANSITION FROM Turn_Off_3 TO P3
    := NOT P3_Led OR NOT UpDeck3Vis_ OR NOT DownDeck3Vis_;
END_TRANSITION
TRANSITION FROM P3 TO Ready
    := Stop;
END_TRANSITION
STEP P4:
    P4_active(N);  // step action
END_STEP
TRANSITION FROM P4 TO Turn_Off_4
    := Current_Deck = 3 AND Served;
END_TRANSITION
STEP Turn_Off_4:
    Turn_Off_4_active(N);  // step action
END_STEP
TRANSITION FROM Turn_Off_4 TO P4
    := NOT P4_Led OR NOT UpDeck4Vis_ OR NOT DownDeck4Vis_;
END_TRANSITION
TRANSITION FROM P4 TO Ready
    := Stop;
END_TRANSITION
STEP P5:
    P5_active(N);  // step action
END_STEP
TRANSITION FROM P5 TO Turn_Off_5
    := Current_Deck = 4 AND Served;
END_TRANSITION
STEP Turn_Off_5:
    Turn_Off_5_active(N);  // step action
END_STEP
TRANSITION FROM Turn_Off_5 TO P5
    := NOT P5_Led OR NOT UpDeck5Vis_ OR NOT DownDeck5Vis_;
END_TRANSITION
TRANSITION FROM P5 TO Ready
    := Stop;
END_TRANSITION
STEP P6:
    P6_active(N);  // step action
END_STEP
TRANSITION FROM P6 TO Turn_Off_6
    := Current_Deck = 5 AND Served;
END_TRANSITION
STEP Turn_Off_6:
    Turn_Off_6_active(N);  // step action
END_STEP
TRANSITION FROM Turn_Off_6 TO P6
    := NOT P6_Led OR NOT UpDeck6Vis_ OR NOT DownDeck6Vis_;
END_TRANSITION
TRANSITION FROM P6 TO Ready
    := Stop;
END_TRANSITION
STEP P7:
    P7_active(N);  // step action
END_STEP
TRANSITION FROM P7 TO Turn_Off_7
    := Current_Deck = 6 AND Served;
END_TRANSITION
STEP Turn_Off_7:
    Turn_Off_7_active(N);  // step action
END_STEP
TRANSITION FROM Turn_Off_7 TO P7
    := NOT P7_Led OR NOT DownDeck7Vis_;
END_TRANSITION
TRANSITION FROM P7 TO Ready
    := Stop;
END_TRANSITION

ACTION Turn_Off_5_active:
P5_Led := FALSE;
UpDeck5Vis_:=FALSE;
DownDeck5Vis_:=FALSE;
END_ACTION

ACTION Refresh_dim_log_exit:

END_ACTION

ACTION P5_exit:
P5_Led := FALSE;
END_ACTION

ACTION Turn_Off_1_active:
P1_Led := FALSE;
UpDeck1Vis_:=FALSE;
DownDeck1Vis_:=FALSE;
END_ACTION

ACTION P2_active:
IF	P2_ AND NOT P2_Led AND Current_Deck <>1 THEN
	P2_Led := TRUE;
	Destination_Deck [i] := 1;
	i := i+1;
END_IF;

IF UpDeck2_ AND NOT UpDeck2Vis_ THEN
	UpDeck2Vis_ := TRUE;
	Up_Calls [ext] := 1;
	Down_Calls [ext] :=8;
	ext := ext +1;
END_IF

IF DownDeck2_ AND NOT DownDeck2Vis_ THEN 
	DownDeck2Vis_ := TRUE;
	Down_Calls [ext] := 1;
	Up_Calls [ext] := 8;
	ext := ext +1;
END_IF
END_ACTION

ACTION P7_exit:
P7_Led := FALSE;
END_ACTION

ACTION Destination_Update_exit:
i := i-1;
Served := FALSE;
END_ACTION

ACTION Turn_Off_6_active:
P6_Led := FALSE;
UpDeck6Vis_:=FALSE;
DownDeck6Vis_:=FALSE;
END_ACTION

ACTION P3_exit:
P3_Led := FALSE;
END_ACTION

ACTION Destination_OUT_active:

END_ACTION

ACTION Wait_TIME_active:
IF PG_ OR P1_ OR P2_ OR P3_ OR P4_ OR P5_ OR P6_ OR P7_ THEN
	Pressed_Start := TRUE;
END_IF

IF UpDeckG_ OR UpDeck1_ OR UpDeck2_ OR UpDeck3_ OR UpDeck4_ OR UpDeck5_ OR UpDeck5_ OR UpDeck6_ THEN
	Pressed_Start := TRUE;
END_IF

IF DownDeck1_ OR DownDeck2_ OR DownDeck3_ OR DownDeck4_ OR DownDeck5_ OR DownDeck6_ OR DownDeck7_ THEN
	Pressed_Start := TRUE;
END_IF
END_ACTION

ACTION Ready_active:
State := 'Ready';
END_ACTION

ACTION Ready_exit:
Doing_What := 'Call_Management';
END_ACTION

ACTION P7_active:
IF	P7_ AND NOT P7_Led AND Current_Deck <>6 THEN
	P7_Led := TRUE; 
	Destination_Deck [i] := 6;
	i := i+1;
END_IF;

IF DownDeck7_ AND NOT DownDeck7Vis_ THEN
	DownDeck7Vis_ := TRUE;
	Down_Calls [ext] := 6;
	Up_Calls [ext] := 8;
	ext := ext +1;
END_IF
END_ACTION

ACTION Turn_Off_G_active:
PG_Led := FALSE;
UpDeckGvis_:=FALSE;
END_ACTION

ACTION WAIT_active:
State := 'Call Management';

IF PG_Led OR P1_Led OR P2_Led OR P3_Led OR P4_Led OR P5_Led OR P6_Led OR P7_Led THEN
	Pressed_Start := TRUE;
END_IF

IF UpDeckGVis_ OR UpDeck1Vis_ OR UpDeck2Vis_ OR UpDeck3Vis_ OR UpDeck4Vis_ OR UpDeck5Vis_ OR UpDeck5Vis_ OR UpDeck6Vis_ THEN
	Pressed_Start := TRUE;
END_IF

IF DownDeck1Vis_ OR DownDeck2Vis_ OR DownDeck3Vis_ OR DownDeck4Vis_ OR DownDeck5Vis_ OR DownDeck6Vis_ OR DownDeck1Vis_ THEN
	Pressed_Start := TRUE;
END_IF
END_ACTION

ACTION PG_active:
IF PG_ AND NOT PG_Led AND Current_Deck <>-1 THEN
	PG_Led := TRUE;
	Destination_Deck [i] := -1;
	i := i+1;
END_IF;

IF UpDeckG_ AND NOT UpDeckGVis_ THEN
	UpDeckGVis_ := TRUE;
	Up_Calls [ext] := -1;
	Down_Calls [ext] := 8;
	ext := ext + 1;
END_IF
END_ACTION

ACTION Can_Go_active:
IF Destination_Deck [0] <> 8 THEN State := 'Can_Go'; END_IF
END_ACTION

ACTION P5_active:
IF	P5_ AND NOT P5_Led AND Current_Deck <>4 THEN 
	P5_Led := TRUE;
	Destination_Deck [i] := 4;
	i := i+1;
END_IF;

IF UpDeck5_ AND NOT UpDeck5Vis_ THEN
	UpDeck5Vis_ := TRUE;
	Up_Calls [ext] := 4;
	Down_Calls [ext] := 8;
	ext := ext +1;
END_IF

IF DownDeck5_ AND NOT DownDeck5Vis_ THEN
	DownDeck5Vis_ := TRUE;
	Down_Calls [ext] := 4;
	Up_Calls [ext] := 8;
	ext := ext +1;
END_IF
END_ACTION

ACTION Sorting_Int_entry:

END_ACTION

ACTION Turn_Off_7_active:
P7_Led := FALSE;
DownDeck7Vis_:=FALSE;
END_ACTION

ACTION P6_exit:
P6_Led := FALSE;
END_ACTION

ACTION P6_active:
(*IF	P6_  AND NOT P6_Led AND Current_Deck <>5 THEN
	P6_Led := TRUE;
	IF ( Destination_Deck[0] - Current_Deck <=0  AND Destination_Deck [0] <> 8 ) THEN
		IF ( Destination_Deck [0] <= 6 AND Current_Deck >=6 ) THEN
			FOR  g:= i-1 TO 0 DO (*Crea lo spazio*)
				Destination_Deck [g+1] := Destination_Deck [g];
			END_FOR
			Destination_Deck [0] := 5;
			ELSE  Destination_Deck [i] := 5;
		END_IF
	END_IF
	IF ( Destination_Deck[0] - Current_Deck >=0  AND Destination_Deck [0] <> 8 ) THEN
		IF ( Destination_Deck [0] >= 6 AND Current_Deck <=6 ) THEN
			
			FOR  g:= i-1 TO 0 DO (*Crea lo spazio*)
				Destination_Deck [g+1] := Destination_Deck [g];
			END_FOR
			Destination_Deck [0] := 5;
			ELSE  Destination_Deck [i] := 5;
			
		END_IF
	END_IF
	i := i+1;
END_IF*)

IF 	P6_ AND NOT P6_Led AND Current_Deck <>5 THEN
	P6_Led := TRUE;
	Destination_Deck [i] := 5;
	i := i+1; 
END_IF;

IF UpDeck6_ AND NOT UpDeck6Vis_ THEN 
	UpDeck6Vis_ := TRUE;
	Up_Calls [ext] := 5;
	Down_Calls [ext] := 8;
	ext := ext +1;
END_IF

IF DownDeck6_ AND NOT DownDeck6Vis_ THEN
	DownDeck6Vis_ := TRUE;
	Down_Calls [ext] := 5;
	Up_Calls [ext] := 8;
	ext := ext +1;
END_IF
END_ACTION

ACTION Turn_Off_2_active:
P2_Led := FALSE;
UpDeck2Vis_:=FALSE;
DownDeck2Vis_:=FALSE;
END_ACTION

ACTION P2_exit:
P2_Led := FALSE;
END_ACTION

ACTION Turn_Off_4_active:
P4_Led := FALSE;
UpDeck4Vis_:=FALSE;
DownDeck4Vis_:=FALSE;
END_ACTION

ACTION Wait_Start_active:

END_ACTION

ACTION Waiting_Int_active:
IF PG_Led OR P1_Led OR P2_Led OR P3_Led OR P4_Led OR P5_Led OR P6_Led OR P7_Led THEN
	Pressed_Int := TRUE;
	ELSE Pressed_Int := FALSE;
END_IF
END_ACTION

ACTION P1_exit:
P1_Led := FALSE;
END_ACTION

ACTION Wait_TIME_entry:
Pressed_Start := FALSE;
END_ACTION

ACTION P3_active:
IF	P3_  AND NOT P3_Led AND Current_Deck <>2 THEN 
	P3_Led := TRUE;
	Destination_Deck [i] := 2;
	i := i+1;
END_IF;

IF UpDeck3_ AND NOT UpDeck3Vis_ THEN
	UpDeck3Vis_ := TRUE;
	Up_Calls [ext] := 2;
	Down_Calls [ext] := 8;
	ext := ext +1;
END_IF

IF DownDeck3_ AND NOT DownDeck3Vis_ THEN 
	DownDeck3Vis_ := TRUE;
	Down_Calls [ext] := 2;
	Up_Calls [ext] := 8;
	ext := ext +1;
END_IF
END_ACTION

ACTION Destination_Update_active:
FOR k := 0 TO i-1 DO
			Destination_Deck [k] := Destination_Deck [k+1];
END_FOR
END_ACTION

ACTION P1_active:
IF 	P1_ AND NOT P1_Led AND Current_Deck <>0 THEN
	P1_Led := TRUE;
	Destination_Deck [i] := 0;
	i := i+1; 
END_IF;
	
IF UpDeck1_ AND NOT UpDeck1Vis_ THEN 
	UpDeck1Vis_ := TRUE;
	Up_Calls [ext] := 0;
	Down_Calls [ext] := 8;
	ext := ext + 1;
END_IF

IF DownDeck1_ AND NOT DownDeck1Vis_ THEN 
	DownDeck1Vis_ := TRUE;
	Down_Calls [ext] := 0;
	Up_Calls [ext] := 8;
	ext := ext +1;
END_IF
END_ACTION

ACTION P4_active:
IF	P4_  AND NOT P4_Led AND Current_Deck <>3 THEN
	P4_Led := TRUE;
	Destination_Deck [i] := 3;
	i := i+1;
END_IF;

IF UpDeck4_ AND NOT UpDeck4Vis_ THEN 
	UpDeck4Vis_ := TRUE;
	Up_Calls [ext] := 3;
	Down_Calls [ext] := 8;
	ext := ext +1;
END_IF

IF DownDeck4_ AND NOT DownDeck4Vis_ THEN 
	DownDeck4Vis_ := TRUE;
	Down_Calls [ext] := 3;
	Up_Calls [ext] := 8;
	ext := ext +1;
END_IF
END_ACTION

ACTION Turn_Off_3_active:
P3_Led := FALSE;
UpDeck3Vis_:=FALSE;
DownDeck3Vis_:=FALSE;
END_ACTION

ACTION P4_exit:
P4_Led := FALSE;
END_ACTION

ACTION Refresh_dim_log_active:
dim_cabin := i;
END_ACTION

ACTION Turn_Off_Leds_active:

CASE ( Current_Deck ) OF
	-1 : IF (NOT PG_Led AND NOT UpDeckGVis_) THEN Turned_Off :=TRUE; END_IF
	 0 : IF (NOT P1_Led AND NOT UpDeck1Vis_ AND NOT DownDeck1Vis_) THEN Turned_Off :=TRUE; END_IF 
	 1 : IF (NOT P2_Led AND NOT UpDeck2Vis_ AND NOT DownDeck2Vis_) THEN Turned_Off :=TRUE; END_IF 
	 2 : IF (NOT P3_Led AND NOT UpDeck3Vis_ AND NOT DownDeck3Vis_) THEN Turned_Off :=TRUE; END_IF 
	 3 : IF (NOT P4_Led AND NOT UpDeck4Vis_ AND NOT DownDeck4Vis_) THEN Turned_Off :=TRUE; END_IF 
	 4 : IF (NOT P5_Led AND NOT UpDeck5Vis_ AND NOT DownDeck5Vis_) THEN Turned_Off :=TRUE; END_IF 
	 5 : IF (NOT P6_Led AND NOT UpDeck6Vis_ AND NOT DownDeck6Vis_) THEN Turned_Off :=TRUE; END_IF 
	 6 : IF (NOT P7_Led AND NOT DownDeck7Vis_) THEN Turned_Off :=TRUE; END_IF  
END_CASE
END_ACTION

ACTION Turn_Off_Leds_exit:
Turned_Off := FALSE;
END_ACTION

ACTION Sorting_Int_active:
dim_cabin := i;

IF ( dim_cabin > 1 ) THEN (*Ordino solo se c'è più di un piano ovviamente*)
	WHILE ( dim_cabin > 1 AND NOT Sorted) DO 
	Sorted := TRUE; 
		FOR j:=0 TO dim_cabin-1 DO
			IF ( ABS ( Destination_Deck [j] - Current_Deck ) >= ABS (Destination_Deck [j+1] - Current_Deck) AND Destination_Deck [j] <> 8 AND Destination_Deck [j+1] <>8 ) THEN
				t := Destination_Deck [j+1];
				Destination_Deck [j+1] := Destination_Deck [j];
				Destination_Deck[j] := t;
				Sorted := FALSE;
			END_IF 
		END_FOR
		dim_cabin := dim_cabin -1;
	END_WHILE
ELSE Sorted := TRUE ; (*Se c'è solo un'elemento è come se fosse gia ordinato*)

END_IF
END_ACTION

ACTION Sorting_Int_exit:
IF (Sorted = TRUE) THEN Sorted := FALSE; END_IF
END_ACTION

ACTION Waiting_Ext_active:

END_ACTION

ACTION Waiting_Int_entry:
Pressed_Int := FALSE;
END_ACTION

ACTION WAIT_entry:
Pressed_Start := FALSE;
END_ACTION

ACTION Turn_Off_3_exit:
P3_ := FALSE;
UpDeck3_ := FALSE;
DownDeck3_ := FALSE;
END_ACTION

ACTION Sorting_Ext_entry:

END_ACTION

ACTION Sorting_Ext_active:

(*Se sto salendo scansiono l'array di discesa per trovare chiamate congruenti*)

IF (Destination_Deck[0] - Current_Deck <=0  AND Destination_Deck [0] <> 8 AND NOT Served) THEN (*Sto scendendo*)
		FOR z:=0 TO 13 DO (*Trovo la posizione della chiamata candidata congruente*)
			IF (( Down_Calls [z] >= Destination_Deck [0] AND Down_Calls [z] <= Current_Deck) (*Deve essere congruente z*)  AND 
				(NOT ( Down_Calls [z+1] >= Destination_Deck [0] AND Down_Calls [z+1] <= Current_Deck) (*Se quella dopo non è congruente prendo z come candidato*) 
					OR ( Down_Calls [z] - Current_Deck < Down_Calls [z+1] - Current_Deck ) (*Se quella dopo ha distanza maggiore la prendo dopo*)
					OR Down_Calls [z+1] = 8 )) THEN
				Position_Ext := z;
			END_IF 
		END_FOR
		IF (Position_Ext <> 8 AND Destination_Deck [0] <> Down_Calls [Position_Ext] (*Non l'ho già inserito*)) THEN
				FOR  z:= i-1 TO 0 DO (*Crea lo spazio*)
					Destination_Deck [z+1] := Destination_Deck [z];
				END_FOR
				i := i+1 ; (*Allargo l'array*)
				Destination_Deck [0] := Down_Calls [Position_Ext]; (* Metto la chiamata esterna nella destinazione *) 
				Down_Calls [Position_Ext] := 8; (*Tolgo la call da Down_Calls mettendoci un 8 al suo posto*)
				Position_Ext := 8; (*Se l'ho inserito allora rimetto a 8 la posizione*)
		END_IF
END_IF



(*Se sto scendendo scansiono l'array di salita per trovare chiamate congruenti*)

IF (Destination_Deck[0] - Current_Deck >= 0 AND Destination_Deck [0] <> 8 AND NOT Served) THEN (*Sto salendo*) 
			FOR z:=0 TO 13 DO
				IF (Up_Calls [z] <= Destination_Deck [0] AND Up_Calls [z] >= Current_Deck  AND 
					(NOT (Up_Calls [z+1] <= Destination_Deck [0] AND Up_Calls [z+1] >= Current_Deck) 
						OR (Up_Calls [z] - Current_Deck < Up_Calls [z+1] - Current_Deck)
						OR Up_Calls [z+1] = 8)) THEN
					Position_Ext := z;
				END_IF 
			END_FOR
		IF (Position_Ext <> 8 AND Destination_Deck [0] <> Up_Calls [Position_Ext] (*Non l'ho già inserito*)) THEN
				Upgrading := TRUE;
				FOR z := i-1 TO 0 DO (*Crea lo spazio*)
					Destination_Deck [z+1] := Destination_Deck [z];
				END_FOR
				i := i+1; (*Allargo l'array*)
				Destination_Deck [0] := Up_Calls [Position_Ext] ; (* Metto la chiamata esterna nella destinazione *) 
				(*Tolgo la call da Up_Calls mettendoci un 8 al suo posto*)
				Up_Calls [Position_Ext] := 8;
				(*Rimetto la posizione a 8*)
				Position_Ext := 8 ;
				Upgrading := FALSE;
		END_IF
END_IF


(* Se l'ascensore è fermo e non ha destinazioni *)
IF (Destination_Deck[0] = 8 AND NOT Served AND NOT (State = 'Can Go')) THEN

    (* Cerca la prima chiamata valida in Up_Calls *)
    FOR z := 0 TO 13 DO
        IF (Up_Calls[z] <> 8) THEN
            Destination_Deck[0] := Up_Calls[z];
            Up_Calls[z] := 8;         (* Rimuovi la chiamata dall’array *)
            i := i + 1;               (* Aggiunta a Destination_Deck *)
            EXIT;                     (* Fermati alla prima valida *)
        END_IF
    END_FOR

    (* Se non c'era nulla in Up_Calls, guarda Down_Calls *)
    IF (Destination_Deck[0] = 8) THEN
        FOR z := 0 TO 13 DO
            IF (Down_Calls[z] <> 8) THEN
                Destination_Deck[0] := Down_Calls[z];
                Down_Calls[z] := 8;
                i := i + 1;
                EXIT;
            END_IF
        END_FOR
    END_IF

END_IF


(*Scalo degli array UP e DOWN*)


IF (Down_Calls[0] = 8 AND Up_Calls[0] = 8 AND (Up_Calls[1] <> 8 OR Down_Calls[1] <> 8)) THEN

    (* Shift degli array: attenzione al limite 12 *)
    FOR z := 0 TO 12 DO
        Down_Calls[z] := Down_Calls[z+1];
        Up_Calls[z]   := Up_Calls[z+1];
    END_FOR

    (* L'ultimo elemento diventa vuoto *)
    Down_Calls[13] := 8;
    Up_Calls[13]   := 8;

    (* Riduci il numero totale di chiamate *)
    ext := ext - 1;

END_IF
END_ACTION

ACTION Can_Go_exit:
State := 'Working' ;
END_ACTION

ACTION Turn_Off_Leds_entry:
Served := TRUE ;
END_ACTION

ACTION Control_Int_active:
(*Caso discesa*)
IF ( Destination_Deck[0] - Current_Deck <=0  AND Destination_Deck [0] <> 8 ) THEN
	
	IF	(P6_) THEN
 
		IF ( Destination_Deck [0] <= 6 AND Current_Deck >=6 ) THEN
			FOR  g:= i-1 TO 0 DO (*Crea lo spazio*)
				Destination_Deck [g+1] := Destination_Deck [g];
			END_FOR
			
			i := i+1 ;
			
			Destination_Deck [0] := 5;
			
		END_IF
 
	END_IF

END_IF
END_ACTION

ACTION Wait_Passengers_exit:
State := 'Call Management';
END_ACTION

END_FUNCTION_BLOCK

// Device/Application/Visualization
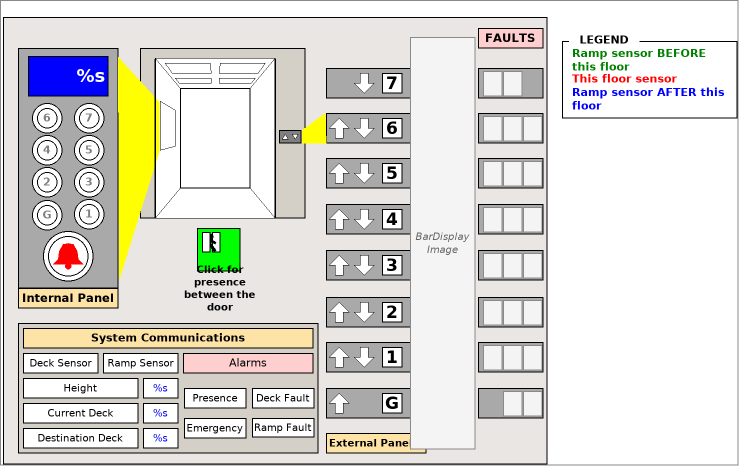
VISUALIZATION Visualization  // 739x466
    Rectangle (3,17 544x447)
    Rectangle (197,228 43x43), colour toggle: GVL.Presence
    Rectangle (18,323 300x130)
    Rectangle (326,433 100x20), "External Panels"
    Rectangle (326,342 100x30)
    Rectangle (382,347 20x20), "1"
    Polygon (354,357) (360,357) (360,347) (368,347) (368,357) (374,357) (364,367), colour toggle: GVL.DownDeck1Vis
        tap GVL.DownDeck1
    Polygon (329,357) (335,357) (335,367) (343,367) (343,357) (349,357) (339,347), colour toggle: GVL.UpDeck1Vis
        tap GVL.UpDeck1
    Rectangle (326,297 100x30)
    Rectangle (382,302 20x20), "2"
    Polygon (354,312) (360,312) (360,302) (368,302) (368,312) (374,312) (364,322), colour toggle: GVL.DownDeck2Vis
        tap GVL.DownDeck2
    Polygon (329,312) (335,312) (335,322) (343,322) (343,312) (349,312) (339,302), colour toggle: GVL.UpDeck2Vis
        tap GVL.UpDeck2
    Rectangle (326,250 100x30)
    Rectangle (382,255 20x20), "3"
    Polygon (354,265) (360,265) (360,255) (368,255) (368,265) (374,265) (364,275), colour toggle: GVL.DownDeck3Vis
        tap GVL.DownDeck3
    Polygon (329,265) (335,265) (335,275) (343,275) (343,265) (349,265) (339,255), colour toggle: GVL.UpDeck3Vis
        tap GVL.UpDeck3
    Rectangle (326,204 100x30)
    Rectangle (382,209 20x20), "4"
    Polygon (354,219) (360,219) (360,209) (368,209) (368,219) (374,219) (364,229), colour toggle: GVL.DownDeck4Vis
        tap GVL.DownDeck4
    Polygon (329,219) (335,219) (335,229) (343,229) (343,219) (349,219) (339,209), colour toggle: GVL.UpDeck4Vis
        tap GVL.UpDeck4
    Rectangle (326,158 100x30)
    Rectangle (382,163 20x20), "5"
    Polygon (354,173) (360,173) (360,163) (368,163) (368,173) (374,173) (364,183), colour toggle: GVL.DownDeck5Vis
        tap GVL.DownDeck5
    Polygon (329,173) (335,173) (335,183) (343,183) (343,173) (349,173) (339,163), colour toggle: GVL.UpDeck5Vis
        tap GVL.UpDeck5
    Rectangle (326,113 100x30)
    Rectangle (382,118 20x20), "6"
    Polygon (354,128) (360,128) (360,118) (368,118) (368,128) (374,128) (364,138), colour toggle: GVL.DownDeck6Vis
        tap GVL.DownDeck6
    Polygon (329,128) (335,128) (335,138) (343,138) (343,128) (349,128) (339,118), colour toggle: GVL.UpDeck6Vis
        tap GVL.UpDeck6
    Rectangle (326,68 100x30)
    Rectangle (382,73 20x20), "7"
    Polygon (354,83) (360,83) (360,73) (368,73) (368,83) (374,83) (364,93), colour toggle: GVL.DownDeck7Vis
        tap GVL.DownDeck7
    Rectangle (326,388 100x30)
    Rectangle (382,393 20x20), "G"
    Polygon (329,403) (335,403) (335,413) (343,413) (343,403) (349,403) (339,393), colour toggle: GVL.UpDeckGVis
        tap GVL.UpDeckG
    RoundedRectangle (18,48 100x240)
    Rectangle (18,288 100x20), "Internal Panel"
    Ellipse (74,199 30x30), colour toggle: GVL.P1Vis
    Ellipse (79,204 20x20), "1"
        tap GVL.P1
    Ellipse (32,200 30x30), colour toggle: GVL.PGVis
    Ellipse (37,205 20x20), "G"
        tap GVL.PG
    Ellipse (74,167 30x30), colour toggle: GVL.P3Vis
    Ellipse (79,172 20x20), "3"
        tap GVL.P3
    Ellipse (32,167 30x30), colour toggle: GVL.P2Vis
    Ellipse (37,172 20x20), "2"
        tap GVL.P2
    Ellipse (74,135 30x30), colour toggle: GVL.P5Vis
    Ellipse (79,140 20x20), "5"
        tap GVL.P5
    Ellipse (32,135 30x30), colour toggle: GVL.P4Vis
    Ellipse (37,140 20x20), "4"
        tap GVL.P4
    Ellipse (74,103 30x30), colour toggle: GVL.P7Vis
    Ellipse (79,108 20x20), "7"
        tap GVL.P7
    Ellipse (32,103 30x30), colour toggle: GVL.P6Vis
    Ellipse (37,108 20x20), "6"
        tap GVL.P6
    Rectangle (28,56 80x40), "%s", text variable: GVL.Destination
    Ellipse (43,231 50x50), tooltip "EMERGENCY", colour toggle: GVL.Emergency
    Group (48,236 40x40)
        toggle GVL.Emergency
        Ellipse (0,0 40x40), tooltip "EMERGENCY"
        Polygon (5,28) (10,23) (11,15) (15,8) (20,7) (25,8) (29,15) (30,23) (35,28)
        Ellipse (17,27 6x6)
    Polygon (35,72) (45,62) (55,72), colour toggle: GVL.Motor_on AND GVL.Up
    Polygon (35,80) (45,90) (55,80), colour toggle: GVL.Motor_on AND NOT GVL.Up
    Group (140,48 165x170)
        Rectangle (0,0 165x170)
        Rectangle (15,10 120x160)
        Polygon (40,40) (15,10) (135,10) (110,40)
        Rectangle (40,40 70x100)
        Polygon (15,170) (40,140) (110,140) (135,170)
        Polygon (20,102) (20,53) (35,62) (35,98)
        Polygon (79,35) (79,30) (115,30) (111,35)
        Polygon (39,35) (35,30) (71,30) (71,35)
        Polygon (32,25) (25,15) (70,15) (71,25)
        Polygon (79,25) (80,15) (125,15) (118,25)
        Group (139,82 22x13)
            Rectangle (0,0 22x13)
            Polygon (3,9) (6,4) (9,9)
            Polygon (13,4) (16,9) (19,4)
    BarDisplayImage (410,37 65x412), value: GVL.Height, style: BarDisplayImage-Gray, scale format: %.0f, scale -20..160
        p3451962224: VisuNativeControl.IP_Offline.Browser
    Rectangle (478,68 65x30)
    Rectangle (478,342 65x30)
    Rectangle (478,297 65x30)
    Rectangle (478,250 65x30)
    Rectangle (478,204 65x30)
    Rectangle (478,158 65x30)
    Rectangle (478,113 65x30)
    Rectangle (478,388 65x30)
    RockerSwitch (483,345 19x25), variable: GVL.Ramp1Down, behaviour: TOGGLE, style: Switch-RockerSwitch-Green
    RockerSwitch (503,345 19x25), variable: GVL.Sensor1, behaviour: TOGGLE, style: Switch-RockerSwitch-Red
    RockerSwitch (523,345 19x25), variable: GVL.Ramp1Up, behaviour: TOGGLE, style: Switch-RockerSwitch-Blue
    RockerSwitch (483,300 19x25), variable: GVL.Ramp2Down, behaviour: TOGGLE, style: Switch-RockerSwitch-Green
    RockerSwitch (503,300 19x25), variable: GVL.Sensor2, behaviour: TOGGLE, style: Switch-RockerSwitch-Red
    RockerSwitch (523,300 19x25), variable: GVL.Ramp2Up, behaviour: TOGGLE, style: Switch-RockerSwitch-Blue
    RockerSwitch (483,253 19x25), variable: GVL.Ramp3Down, behaviour: TOGGLE, style: Switch-RockerSwitch-Green
    RockerSwitch (503,253 19x25), variable: GVL.Sensor3, behaviour: TOGGLE, style: Switch-RockerSwitch-Red
    RockerSwitch (523,253 19x25), variable: GVL.Ramp3Up, behaviour: TOGGLE, style: Switch-RockerSwitch-Blue
    RockerSwitch (483,207 19x25), variable: GVL.Ramp4Down, behaviour: TOGGLE, style: Switch-RockerSwitch-Green
    RockerSwitch (503,207 19x25), variable: GVL.Sensor4, behaviour: TOGGLE, style: Switch-RockerSwitch-Red
    RockerSwitch (523,207 19x25), variable: GVL.Ramp4Up, behaviour: TOGGLE, style: Switch-RockerSwitch-Blue
    RockerSwitch (483,161 19x25), variable: GVL.Ramp5Down, behaviour: TOGGLE, style: Switch-RockerSwitch-Green
    RockerSwitch (503,161 19x25), variable: GVL.Sensor5, behaviour: TOGGLE, style: Switch-RockerSwitch-Red
    RockerSwitch (523,161 19x25), variable: GVL.Ramp5Up, behaviour: TOGGLE, style: Switch-RockerSwitch-Blue
    RockerSwitch (483,116 19x25), variable: GVL.Ramp6Down, behaviour: TOGGLE, style: Switch-RockerSwitch-Green
    RockerSwitch (503,116 19x25), variable: GVL.Sensor6, behaviour: TOGGLE, style: Switch-RockerSwitch-Red
    RockerSwitch (523,116 19x25), variable: GVL.Ramp6Up, behaviour: TOGGLE, style: Switch-RockerSwitch-Blue
    RockerSwitch (483,71 19x25), variable: GVL.Ramp7Down, behaviour: TOGGLE, style: Switch-RockerSwitch-Green
    RockerSwitch (503,71 19x25), variable: GVL.Sensor7, behaviour: TOGGLE, style: Switch-RockerSwitch-Red
    RockerSwitch (503,391 19x25), variable: GVL.SensorG, behaviour: TOGGLE, style: Switch-RockerSwitch-Red
    RockerSwitch (523,391 19x25), variable: GVL.RampGUp, behaviour: TOGGLE, style: Switch-RockerSwitch-Blue
    Rectangle (478,28 65x20), "FAULTS"
    Polygon (302,130) (325,113) (326,143) (302,143), invisible if: (GVL.Closing OR GVL.Opening) OR GVL.Closed
    Polygon (118,57) (159,102) (159,151) (119,279), invisible if: (GVL.Closing OR GVL.Opening) OR GVL.Closed
    Rectangle (155,58 0x160)
        p3528305787: GVL.Door
    Rectangle (275,58 0x160)
        p3528305787: -GVL.Door
    Rectangle (23,328 290x20), "System Communications"
    Rectangle (183,353 130x20), "Alarms"
    Rectangle (23,353 75x20), "Deck Sensor", colour toggle: GVL.DeckSensor
    Rectangle (143,378 35x20), "%s", text variable: GVL.Height
    Rectangle (184,388 62x20), "Presence", colour toggle: GVL.Presence
    Rectangle (103,353 75x20), "Ramp Sensor", colour toggle: GVL.RampSensor
    Rectangle (143,403 35x20), "%s", text variable: GVL.Current
    Rectangle (143,428 35x20), "%s", text variable: GVL.Destination
    Rectangle (252,388 62x20), "Deck Fault", colour toggle: GVL.FaultSensorAlarm
    Rectangle (184,418 62x20), "Emergency", colour toggle: GVL.EmergencyVis
    Rectangle (252,418 62x19), "Ramp Fault", colour toggle: GVL.FaultRampAlarm
    Rectangle (23,378 115x20), "Height"
    Rectangle (23,403 115x20), "Current Deck"
    Rectangle (23,428 115x20), "Destination Deck"
    Group (562,25 175x93)
        Rectangle (0,16 175x77)
        Rectangle (7,39 160x30), "This floor sensor"
        Rectangle (7,59 160x30), "Ramp sensor AFTER this floor"
        Rectangle (7,0 70x30), "LEGEND"
        Rectangle (7,20 160x30), "Ramp sensor BEFORE this floor"
    Group (202,232 33x34)
        toggle GVL.Presence
        Rectangle (10,0 8x20)
        Polygon (5,10) (12,20) (14,18) (5,6)
        Ellipse (6,2 5x5)
        Polygon (4,8) (13,12) (14,10) (4,4)
        Rectangle (0,0 8x20)
    Rectangle (169,273 102x31), "Click for presence between the door"
END_VISUALIZATION
